# EPICS substitutions: kstar/siteApp/TS2/TS2App/Db/ts_mean_B3.substitutions
#
file db/TS_CH_value.db
{
    pattern
        { DEV,    ID,       TAIL,     DESC,                ARG     }

#
        {"B3",    "0",      "MEAN",   "mean value",    "raw_mean"}
        {"B3",    "1",       "MEAN",   "mean value",    "raw_mean"}
        {"B3",    "2",       "MEAN",   "mean value",    "raw_mean"}
        {"B3",    "3",       "MEAN",   "mean value",    "raw_mean"}
        {"B3",    "4",       "MEAN",   "mean value",    "raw_mean"}
        {"B3",    "5",       "MEAN",   "mean value",    "raw_mean"}
        {"B3",    "6",       "MEAN",   "mean value",    "raw_mean"}
        {"B3",    "7",       "MEAN",   "mean value",    "raw_mean"}
        {"B3",    "8",       "MEAN",   "mean value",    "raw_mean"}
        {"B3",    "9",       "MEAN",   "mean value",    "raw_mean"}
        {"B3",    "10",       "MEAN",   "mean value",    "raw_mean"}
        {"B3",    "11",       "MEAN",   "mean value",    "raw_mean"}
        {"B3",    "12",       "MEAN",   "mean value",    "raw_mean"}
        {"B3",    "13",       "MEAN",   "mean value",    "raw_mean"}
        {"B3",    "14",       "MEAN",   "mean value",    "raw_mean"}
        {"B3",    "15",       "MEAN",   "mean value",    "raw_mean"}
#
#
        {"B3",    "0",      "BG_MEAN",   "background mean value",    "bg_mean"}
        {"B3",    "1",      "BG_MEAN",   "background mean value",    "bg_mean"}
        {"B3",    "2",      "BG_MEAN",   "background mean value",    "bg_mean"}
        {"B3",    "3",      "BG_MEAN",   "background mean value",    "bg_mean"}
        {"B3",    "4",      "BG_MEAN",   "background mean value",    "bg_mean"}
        {"B3",    "5",      "BG_MEAN",   "background mean value",    "bg_mean"}
        {"B3",    "6",      "BG_MEAN",   "background mean value",    "bg_mean"}
        {"B3",    "7",      "BG_MEAN",   "background mean value",    "bg_mean"}
        {"B3",    "8",      "BG_MEAN",   "background mean value",    "bg_mean"}
        {"B3",    "9",      "BG_MEAN",   "background mean value",    "bg_mean"}
        {"B3",    "10",      "BG_MEAN",   "background mean value",    "bg_mean"}
        {"B3",    "11",      "BG_MEAN",   "background mean value",    "bg_mean"}
        {"B3",    "12",      "BG_MEAN",   "background mean value",    "bg_mean"}
        {"B3",    "13",      "BG_MEAN",   "background mean value",    "bg_mean"}
        {"B3",    "14",      "BG_MEAN",   "background mean value",    "bg_mean"}
        {"B3",    "15",      "BG_MEAN",   "background mean value",    "bg_mean"}

}
